{attribute 'linkalways'} 
{attribute 'no_explicit_call' := 'This FB is a CLASS and must be accessed using methods or properties'}
{attribute 'enable_dynamic_creation'}
FUNCTION_BLOCK Node_F_VN_MaxElementElementwise_TcVnVector2_DINT EXTENDS VisionNode
VAR
    ipContainer : _ITcVnContainer;
    aMax : _TcVnVector2_DINT;
    hrPrev : _HRESULT(S_OK);
    hresult : _HRESULT(S_OK);
END_VAR

METHOD PUBLIC  Clone : I_Node
VAR
	pNode : POINTER TO Node_F_VN_MaxElementElementwise_TcVnVector2_DINT;
END_VAR
pNode := __NEW(Node_F_VN_MaxElementElementwise_TcVnVector2_DINT);
Clone := pNode^;
END_METHOD

METHOD FB_init : BOOL
VAR_INPUT
	bInitRetains : BOOL; // if TRUE, the retain variables are initialized (warm start / cold start)
	bInCopyCode : BOOL;  // if TRUE, the instance afterwards gets moved into the copy code (online change)
END_VAR
AddInput('ipContainer', ipContainer);
AddInput('hrPrev', hrPrev);
AddOutput('ipContainer', ipContainer);
AddOutput('aMax', aMax);
AddOutput('hresult',hresult);
END_METHOD

METHOD PROTECTED OnExecute
hresult.Value := F_VN_MaxElementElementwise_TcVnVector2_DINT(
    ipContainer := ipContainer.Value,
    aMax := aMax.Value,
    hrPrev:= hrPrev.Value);
END_METHOD

METHOD PUBLIC PreExecutionCheck
VAR_INPUT
	Check : I_PreExecutionChecks;
END_VAR
Check.IsTrue(ipContainer.IsValid, 'ipContainer must be a valid container');
Check.IsTrue(ipContainer.IsType(TC_GLOBAL_CONST_LIST.ContainerType_Vector_TcVnVector2_DINT), 'ipContainer contains incorrect type');
END_METHOD

END_FUNCTION_BLOCK

(* stored: Version 1.1.0.1, ProductVersion 3.1.4026.13
   POU Node_F_VN_MaxElementElementwise_TcVnVector2_DINT: Id {ec642846-62ca-4507-8dda-de38e72409be}, SpecialFunc None
   Folder Constructor: Id {28beb0ad-93c4-4294-b673-0cc08cd52890}
   Method Clone: Id {7695d4e1-d5c6-4b89-9c59-509f60f6033d}
   Method FB_init: Id {e0c04b11-75cf-4dfe-b7e3-a6c749ba0d76}
   Method OnExecute: Id {98b713bd-d94d-4c96-b35c-da595afe172c}
   Method PreExecutionCheck: Id {9086d9b3-d83c-4796-a1e8-846538413620} *)
